GLOBALCONSTANTS quarter (* Global constants *)
  (* Standard: 61499-1; Description: Copyright (c) 2024 HR Agrartechnik GmbH This program and the accompanying materials are made available under the terms of the Eclipse Public License 2.0 which is available at https://www.eclipse.org/legal/epl-2.0/ SPDX-License-Identifier: EPL-2.0 *)
  (* Version 1.0, 2024-02-23, Franz Höpfinger, HR Agrartechnik GmbH *)
  VAR_GLOBAL CONSTANT
    STATUS_DISABLED : BYTE := 2#00; (* Disabled (off, passive, etc.) *)
    STATUS_ENABLED : BYTE := 2#01; (* Enabled (on, active, etc.) *)
    STATUS_ERROR : BYTE := 2#10; (* Error indicator *)
    STATUS_NOT_AVAILABLE : BYTE := 2#11; (* Not available or not installed *)
    STATUS_DISABLED_msg : STRING := 'Disabled (off, passive, etc.)';
    STATUS_ENABLED_msg : STRING := 'Enabled (on, active, etc.)';
    STATUS_ERROR_msg : STRING := 'Error indicator';
    STATUS_NOT_AVAILABLE_msg : STRING := 'Not available or not installed';
    COMMAND_DISABLE : BYTE := 2#00; (* Command to disable function (turn off, etc.) *)
    COMMAND_ENABLE : BYTE := 2#01; (* Command to enable function (turn on, etc.) *)
    COMMAND_RESERVED : BYTE := 2#10; (* Reserved *)
    COMMAND_NO_ACTION : BYTE := 2#11; (* Don't care/take no action (leave function as is) *)
    COMMAND_DISABLE_msg : STRING := 'Command to disable function (turn off, etc.)';
    COMMAND_ENABLE_msg : STRING := 'Command to enable function (turn on, etc.)';
    COMMAND_RESERVED_msg : STRING := 'Reserved';
    COMMAND_NO_ACTION_msg : STRING := 'Don`t care/take no action (leave function as is)';
  END_VAR
END_GLOBALCONSTANTS
